// SIMATIC S7-200 project (STEP 7-Micro/WIN), CPU 221 REL 01.10

ORGANIZATION_BLOCK 主程序:OB1
TITLE=程序注释
BEGIN
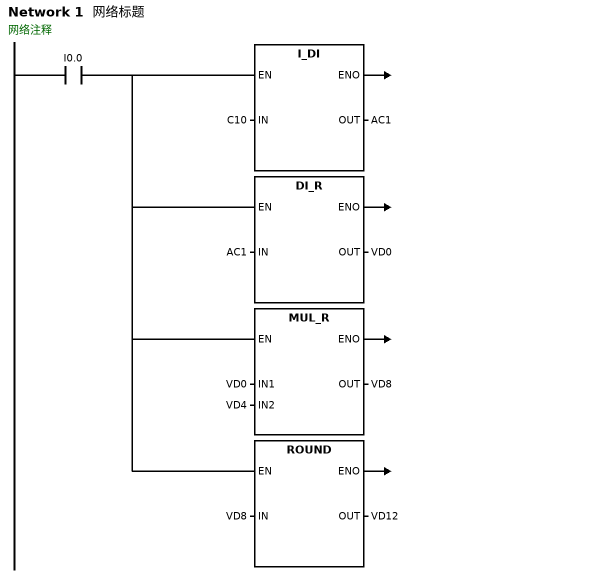
Network 1 // 网络标题
// 网络注释
LD     I0.0
ITD    C10, AC1
DTR    AC1, VD0
MOVR   VD0, VD8
*R     VD4, VD8
ROUND  VD8, VD12
END_ORGANIZATION_BLOCK
